{attribute 'qualified_only'}
{attribute 'strict'}
TYPE E_ModuleState :
(
    MANUAL := 0,   (* Manual mode *)
    AUTO := 1      (* Auto mode *)
);
END_TYPE;

(* stored: Version 1.1.0.1, ProductVersion 3.1.4024.13
   DUT E_ModuleState: Id {770421af-bddf-4caa-ae27-505698416713} *)
